PROGRAM MainProBox
(**************************************************************************************
 * 	Application		:	ProBox
 *	Revision		:	$$
 *	Revision date	:	$$
 *	Last changed by	:	$$
 *	URL				:	$$
 *
 *	Purpose			:	ProBox main application.
 *
 * ------------------------------------------------------------------------------------
 *	Copyright Swisslog [IP AG], Switzerland. All rights reserved.
 * 
 * ------------------------------------------------------------------------------------
 *	
 * 	Revision History: 
 *
 * 	VERSION			DATE			INITIALS			DESCRIPTION
 *	0.1				01.01.2001		swl					Example
 *
 **************************************************************************************)
VAR
	fbHardwareInputs					: FB_HardwareInputs;
	fbHardwareOutputs					: FB_HardwareOutputs;	
	fbSafetyCustomization				: FB_SafetyCompositionCustomized;
END_VAR
VAR_TEMP
BCFisInitiaded:BOOL;
		
END_VAR

 
(*******************************************************************************************************************
  
***************************************************************************************************************)
BCFisInitiaded :=MainConv.Init;

EMULATION_ENABLED := TRUE;
IF(EMULATION_ENABLED) THEN
	MainConvEmulation();
END_IF

IF(BCFisInitiaded) THEN 
	IF(NOT EMULATION_ENABLED) THEN
		// Get HW Inputs
		fbHardwareInputs();
	END_IF		
	// run Custom debug functions
	F_DebugCompositionCustomization();  
END_IF
	
// Custom safety functions 
fbSafetyCustomization(_InitSafety:=BCFisInitiaded AND NOT EMULATION_ENABLED);
//run BCF
MainConv();

//if MainConv is initiated and not emulation enabled
IF(BCFisInitiaded) THEN
	//Set HW Outputs
	fbHardwareOutputs();		
END_IF

END_PROGRAM

(* stored: Version 1.1.0.1, ProductVersion 3.1.4024.9
   POU MainProBox: Id {0516c6bc-8e87-48f5-94c4-5ebe723f98ef}, SpecialFunc None *)
